Fanuc KAREL source: kb00186.KL

PROGRAM KB00186
%NOLOCKGROUP
VAR
P1:REAL;RESULT:REAL
BEGIN
--
P1=1.0
RESULT=SIN(P1)
END KB00186
